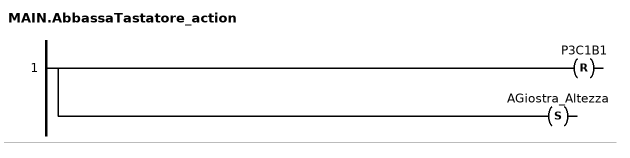
[picture p48: MAIN.AbbassaTastatore_action (LD)]
_LD_ (* Ladder Diagram *)
NETWORK 1
	* --- (R P3C1B1) (S AGiostra_Altezza)
_END_LD_
(* the same logic as Structured Text *)
(* Network 1 *)
P3C1B1 := FALSE;
AGiostra_Altezza := TRUE;
END_ACTION

ACTION SetVarTast2_action:
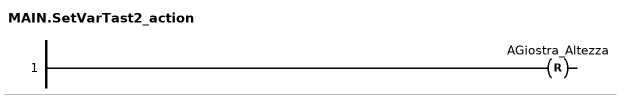
_LD_ (* Ladder Diagram *)
NETWORK 1
	* --- (R AGiostra_Altezza)
_END_LD_
(* the same logic as Structured Text *)
(* Network 1 *)
AGiostra_Altezza := FALSE;
END_ACTION

ACTION ResetL3_action:
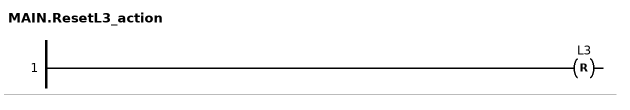
_LD_ (* Ladder Diagram *)
NETWORK 1
	* --- (R L3)
_END_LD_
(* the same logic as Structured Text *)
(* Network 1 *)
L3 := FALSE;
END_ACTION

ACTION Rot6_action:
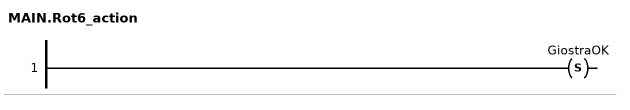
_LD_ (* Ladder Diagram *)
NETWORK 1
	* --- (S GiostraOK)
_END_LD_
(* the same logic as Structured Text *)
(* Network 1 *)
GiostraOK := TRUE;
END_ACTION

ACTION Step100_action:
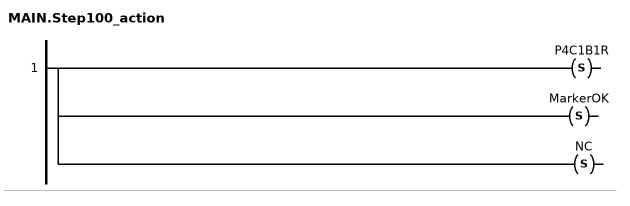
_LD_ (* Ladder Diagram *)
NETWORK 1
	* --- (S P4C1B1R) (S MarkerOK) (S NC)
_END_LD_
(* the same logic as Structured Text *)
(* Network 1 *)
P4C1B1R := TRUE;
MarkerOK := TRUE;
NC := TRUE;
END_ACTION

ACTION SetVarTast3_action:
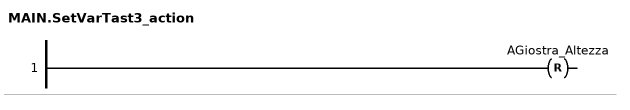
_LD_ (* Ladder Diagram *)
NETWORK 1
	* --- (R AGiostra_Altezza)
_END_LD_
(* the same logic as Structured Text *)
(* Network 1 *)
AGiostra_Altezza := FALSE;
END_ACTION

ACTION UnAltroResetL3_action:
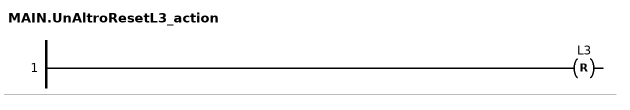
_LD_ (* Ladder Diagram *)
NETWORK 1
	* --- (R L3)
_END_LD_
(* the same logic as Structured Text *)
(* Network 1 *)
L3 := FALSE;
END_ACTION

ACTION Rot7_action:
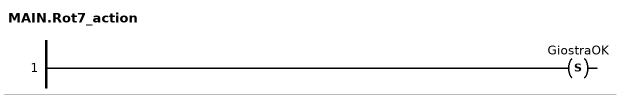
_LD_ (* Ladder Diagram *)
NETWORK 1
	* --- (S GiostraOK)
_END_LD_
(* the same logic as Structured Text *)
(* Network 1 *)
GiostraOK := TRUE;
END_ACTION

ACTION Step99_action:
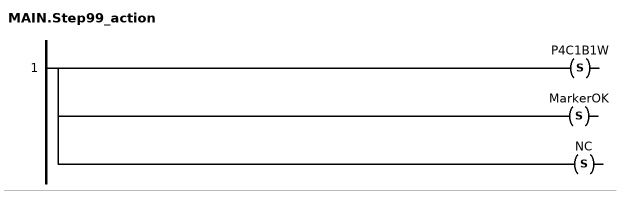
_LD_ (* Ladder Diagram *)
NETWORK 1
	* --- (S P4C1B1W) (S MarkerOK) (S NC)
_END_LD_
(* the same logic as Structured Text *)
(* Network 1 *)
P4C1B1W := TRUE;
MarkerOK := TRUE;
NC := TRUE;
END_ACTION

ACTION SetVarTast_action:
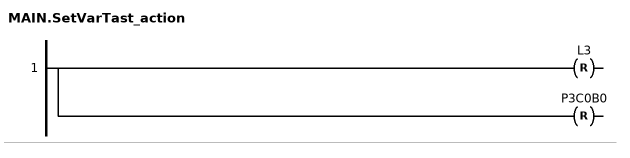
_LD_ (* Ladder Diagram *)
NETWORK 1
	* --- (R L3) (R P3C0B0)
_END_LD_
(* the same logic as Structured Text *)
(* Network 1 *)
L3 := FALSE;
P3C0B0 := FALSE;
END_ACTION

ACTION Rot8_action:
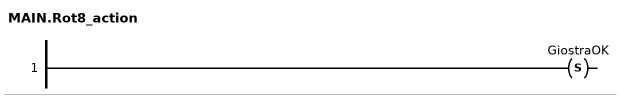
_LD_ (* Ladder Diagram *)
NETWORK 1
	* --- (S GiostraOK)
_END_LD_
(* the same logic as Structured Text *)
(* Network 1 *)
GiostraOK := TRUE;
END_ACTION

ACTION Step98_action:
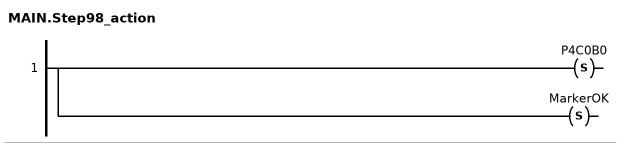
_LD_ (* Ladder Diagram *)
NETWORK 1
	* --- (S P4C0B0) (S MarkerOK)
_END_LD_
(* the same logic as Structured Text *)
(* Network 1 *)
P4C0B0 := TRUE;
MarkerOK := TRUE;
END_ACTION

ACTION ResetMarker_action:
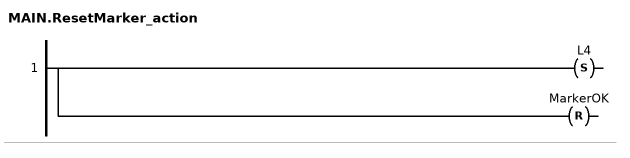
_LD_ (* Ladder Diagram *)
NETWORK 1
	* --- (S L4) (R MarkerOK)
_END_LD_
(* the same logic as Structured Text *)
(* Network 1 *)
L4 := TRUE;
MarkerOK := FALSE;
END_ACTION

ACTION Step81_action:
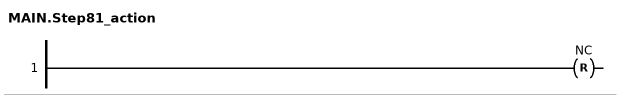
_LD_ (* Ladder Diagram *)
NETWORK 1
	* --- (R NC)
_END_LD_
(* the same logic as Structured Text *)
(* Network 1 *)
NC := FALSE;
END_ACTION

ACTION SetVarMarkR_action:
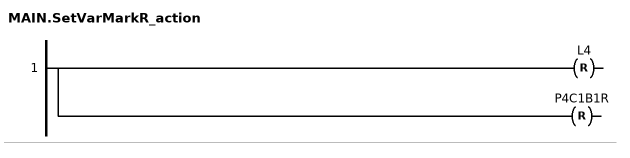
_LD_ (* Ladder Diagram *)
NETWORK 1
	* --- (R L4) (R P4C1B1R)
_END_LD_
(* the same logic as Structured Text *)
(* Network 1 *)
L4 := FALSE;
P4C1B1R := FALSE;
END_ACTION

ACTION Rot11_action:
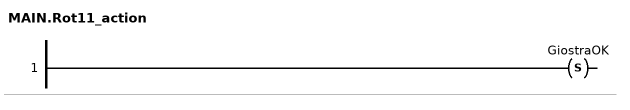
_LD_ (* Ladder Diagram *)
NETWORK 1
	* --- (S GiostraOK)
_END_LD_
(* the same logic as Structured Text *)
(* Network 1 *)
GiostraOK := TRUE;
END_ACTION

ACTION Step95_action:
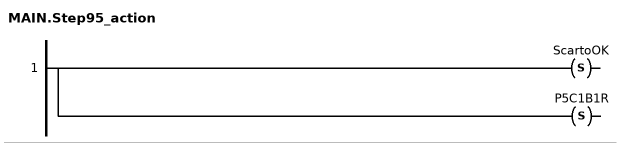
_LD_ (* Ladder Diagram *)
NETWORK 1
	* --- (S ScartoOK) (S P5C1B1R)
_END_LD_
(* the same logic as Structured Text *)
(* Network 1 *)
ScartoOK := TRUE;
P5C1B1R := TRUE;
END_ACTION

ACTION SetVarMark_action:
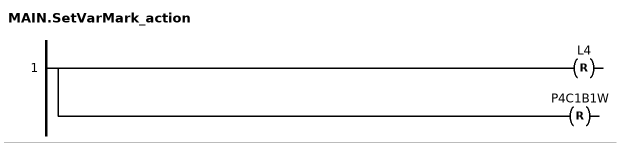
_LD_ (* Ladder Diagram *)
NETWORK 1
	* --- (R L4) (R P4C1B1W)
_END_LD_
(* the same logic as Structured Text *)
(* Network 1 *)
L4 := FALSE;
P4C1B1W := FALSE;
END_ACTION

ACTION Rot10_action:
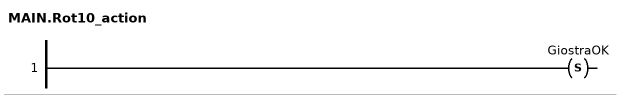
_LD_ (* Ladder Diagram *)
NETWORK 1
	* --- (S GiostraOK)
_END_LD_
(* the same logic as Structured Text *)
(* Network 1 *)
GiostraOK := TRUE;
END_ACTION

ACTION Step96_action:
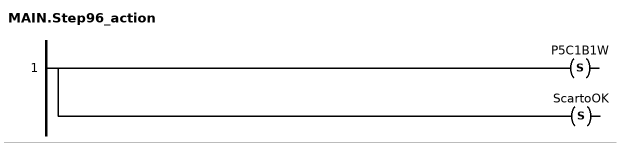
_LD_ (* Ladder Diagram *)
NETWORK 1
	* --- (S P5C1B1W) (S ScartoOK)
_END_LD_
(* the same logic as Structured Text *)
(* Network 1 *)
P5C1B1W := TRUE;
ScartoOK := TRUE;
END_ACTION

ACTION AbbassaMarker_action:
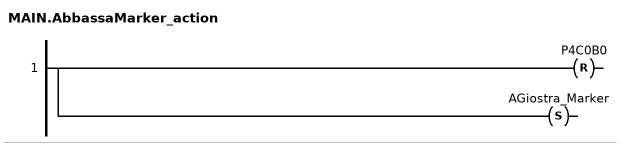
_LD_ (* Ladder Diagram *)
NETWORK 1
	* --- (R P4C0B0) (S AGiostra_Marker)
_END_LD_
(* the same logic as Structured Text *)
(* Network 1 *)
P4C0B0 := FALSE;
AGiostra_Marker := TRUE;
END_ACTION

ACTION Step93_action:
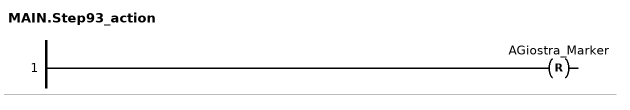
_LD_ (* Ladder Diagram *)
NETWORK 1
	* --- (R AGiostra_Marker)
_END_LD_
(* the same logic as Structured Text *)
(* Network 1 *)
AGiostra_Marker := FALSE;
END_ACTION

ACTION ResetL4_action:
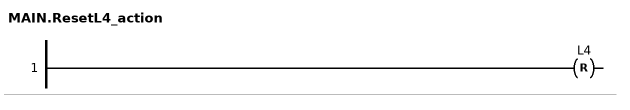
_LD_ (* Ladder Diagram *)
NETWORK 1
	* --- (R L4)
_END_LD_
(* the same logic as Structured Text *)
(* Network 1 *)
L4 := FALSE;
END_ACTION

ACTION Rot9_action:
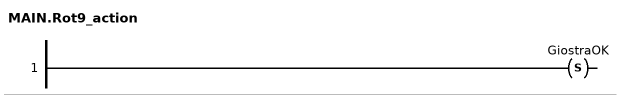
_LD_ (* Ladder Diagram *)
NETWORK 1
	* --- (S GiostraOK)
_END_LD_
(* the same logic as Structured Text *)
(* Network 1 *)
GiostraOK := TRUE;
END_ACTION

ACTION Step97_action:
